{attribute 'qualified_only'}
VAR_GLOBAL
END_VAR

(* stored: Version 1.1.0.1, ProductVersion 3.1.4022.7
   GVL GVL_06_Output_Servo_Motor_Shelf_Y: Id {4697f004-25c8-4868-97c1-e6295f6dfcb8} *)
